TYPE "CTrk_Log"
VERSION : 0.1
// Block: CTrk_Log
   STRUCT
      DataValid : Bool;
      MES_Received : Bool;
      MES_Send : Bool;
      Logger_Send : Bool;
      O_ID : DInt;
      Diameter : Real;
      Tickness : Real;
      "Tickness_Out-Of-Tol" : Bool;
      DT : DTL;
   END_STRUCT;

END_TYPE
